% RSLogix 500 project INTRO TO PLC - JOB 14.RSS, saved by version 10.00.00.00 %
PROJECT "PL06B"    % processor: Bul.1763 MicroLogix 1100 Series B %

PROGRAM FILES
  LAD 2   6 rungs

DATA FILES
  O0 OUTPUT  4 elements
  I1 INPUT  6 elements
  S2 STATUS  66 elements
  B3 BINARY  1 elements
  T4 TIMER  2 elements
  C5 COUNTER  2 elements
  R6 CONTROL  1 elements
  N7 INTEGER  1 elements
  F8 FLOAT  1 elements

LADDER 2
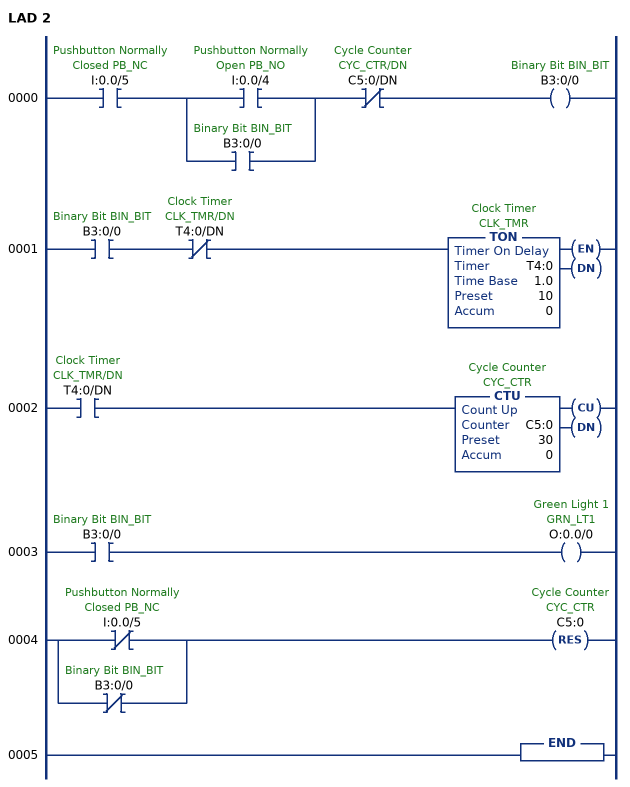
% Rung: 0 %
SOR XIC I:0.0/5 BST XIC I:0.0/4 NXB XIC B3:0/0 BND XIO C5:0/DN OTE B3:0/0 EOR
%   I:0.0/5  PB_NC  "Pushbutton Normally Closed" %
%   I:0.0/4  PB_NO  "Pushbutton Normally Open" %
%   B3:0/0  BIN_BIT  "Binary Bit" %
%   C5:0  CYC_CTR  "Cycle Counter" %
% Rung: 1 %
SOR XIC B3:0/0 XIO T4:0/DN TON T4:0 1.0 10 0 EOR
%   B3:0/0  BIN_BIT  "Binary Bit" %
%   T4:0  CLK_TMR  "Clock Timer" %
% Rung: 2 %
SOR XIC T4:0/DN CTU C5:0 30 0 EOR
%   T4:0  CLK_TMR  "Clock Timer" %
%   C5:0  CYC_CTR  "Cycle Counter" %
% Rung: 3 %
SOR XIC B3:0/0 OTE O:0.0/0 EOR
%   B3:0/0  BIN_BIT  "Binary Bit" %
%   O:0.0/0  GRN_LT1  "Green Light 1" %
% Rung: 4 %
SOR BST XIO I:0.0/5 NXB XIO B3:0/0 BND RES C5:0 EOR
%   I:0.0/5  PB_NC  "Pushbutton Normally Closed" %
%   B3:0/0  BIN_BIT  "Binary Bit" %
%   C5:0  CYC_CTR  "Cycle Counter" %
% Rung: 5 %
SOR END EOR

OTHER DOCUMENTED ADDRESSES
  B3:0/1  SEAL2  "Seal 2"
  C5:1  CYC_CTR2  "Cycle Counter 2"
  I:0.0/0  SS1A  "Selector Switch 1 Position A"
  I:0.0/1  SS1B  "Selector Switch 1 Position B"
  I:0.0/2  SS2A  "Selector Switch 2 Position A"
  I:0.0/3  SS2B  "Selector Switch 2 Position B"
  O:0.0/1  RED_LT  "Red Light"
  O:0.0/2  YLW_LT  "Yellow Light"
  O:0.0/3  GRN_LT2  "Green Light 2"
  T4:1  LT_TMR2  "Light Timer 2"

COMMENTS NOT ATTACHED TO A CURRENT RUNG
  T4:1: Same Logic without using Binary Bits

DATA TABLE (non-zero values as saved)
DATA T4
% .PRE .ACC %
% T4:0 % 10 0
% T4:1 % 10 0
DATA C5
% .PRE .ACC %
% C5:0 % 30 0
% C5:1 % 5 5
